FUNCTION_BLOCK QW
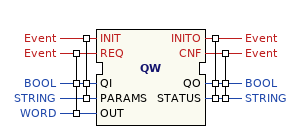
  EVENT_INPUT
    INIT WITH QI, PARAMS;
    REQ WITH QI, OUT;
  END_EVENT
  EVENT_OUTPUT
    INITO WITH QO, STATUS;
    CNF WITH QO, STATUS;
  END_EVENT
  VAR_INPUT
    QI : BOOL;
    PARAMS : STRING;
    OUT : WORD;
  END_VAR
  VAR_OUTPUT
    QO : BOOL;
    STATUS : STRING;
  END_VAR
END_FUNCTION_BLOCK
